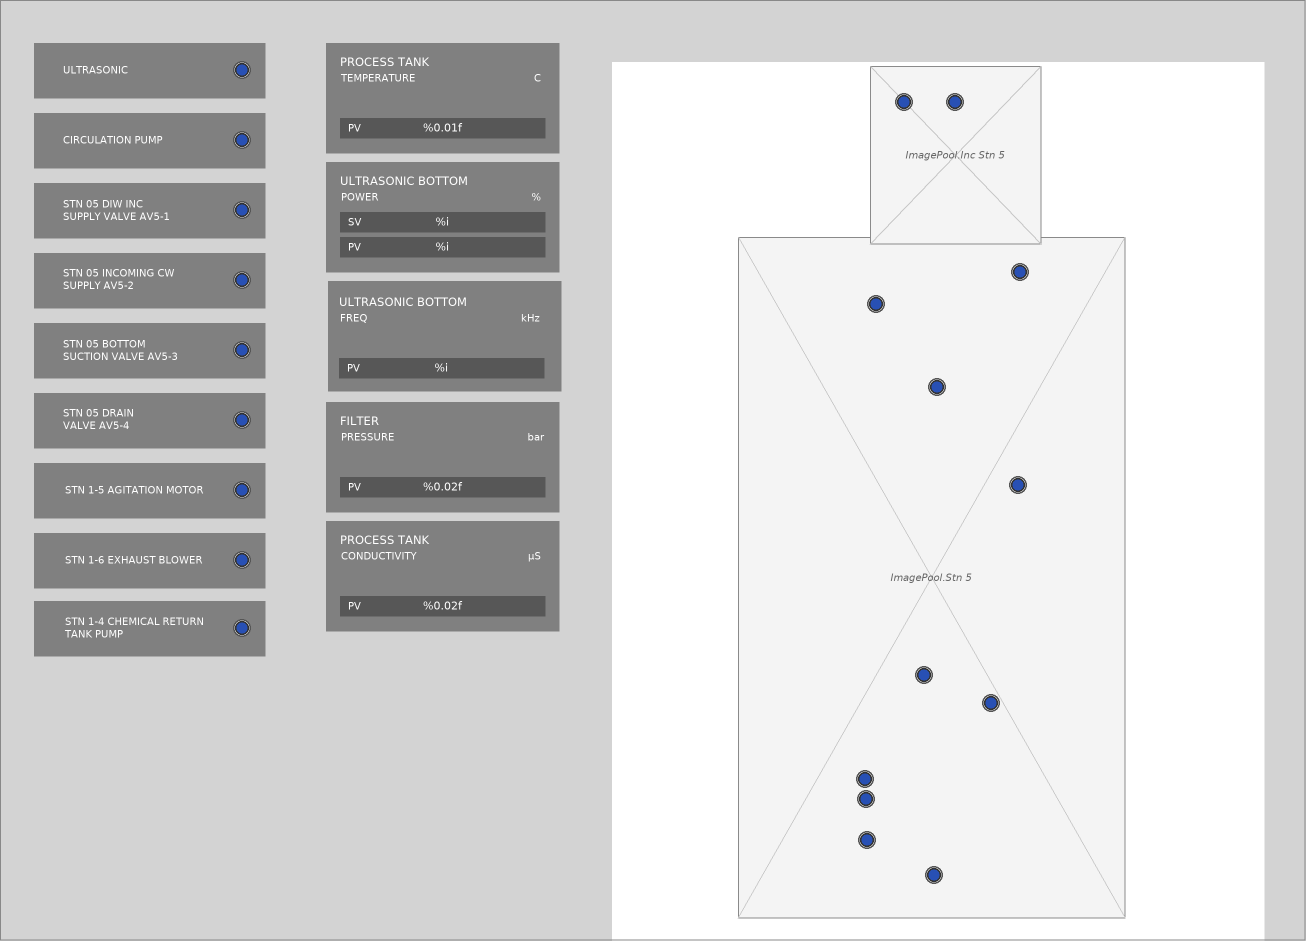
VISUALIZATION Auto_Station05  // 1306x941
    Rectangle (0,0 1306x875)
    RoundedRectangle (34,43 231x55)
    Label (60,62 163x16), "ULTRASONIC"
    Lamp1 (232,60 20x20), variable: ARdsMAP_HmiVariableStn[5].bProTankUsBtm_IND, style: Lamp-Lamp1-Blue
    RoundedRectangle (34,113 231x55)
    Label (60,132 151x16), "CIRCULATION PUMP"
    Lamp1 (232,130 20x20), variable: ARdsMAP_HmiVariableStn[5].bProTankPump_IND, style: Lamp-Lamp1-Blue
    RoundedRectangle (326,43 233x110)
    Label (337,54 150x16), "PROCESS TANK"
    Label (338,67 99x22), "TEMPERATURE"
    Label (515,67 29x22), "C"
    Label (345,92 22x22)
    Rectangle (340,118 205x20), "%0.01f", text variable: ARrStnTempPV[5]
    Label (345,117 22x22), "PV"
    Group (326,162 233x110)
        RoundedRectangle (0,0 233x110)
        Label (11,11 150x16), "ULTRASONIC BOTTOM"
        Label (12,24 99x22), "POWER"
        Label (189,24 29x22), "%"
        Rectangle (14,50 205x20), "%i", text variable: DSWeberEnclosure[1].DSWeberGenerator[3].IN_iTargetPowerPercentSetPoint
        Label (19,49 22x22), "SV"
        Rectangle (14,75 205x20), "%i", text variable: ARiStnUSBtmAPv[5]
        Label (19,74 22x22), "PV"
    RoundedRectangle (326,402 233x110)
    Label (337,413 150x16), "FILTER"
    Label (338,426 99x22), "PRESSURE"
    Label (515,426 32x22), "bar"
    Rectangle (340,477 205x20), "%0.02f", text variable: ARrStnFilterPressurePV[5]
    Label (345,476 22x22), "PV"
    RoundedRectangle (326,521 233x110)
    Label (337,532 150x16), "PROCESS TANK"
    Label (338,545 99x22), "CONDUCTIVITY"
    Label (515,545 29x22), "μS"
    Label (345,570 22x22)
    Rectangle (340,596 205x20), "%0.02f", text variable: ARrStnConductivityPV[5]
    Label (345,595 22x22), "PV"
    RoundedRectangle (328,281 233x110)
    Label (337,307 99x22), "FREQ"
    Label (336,294 150x16), "ULTRASONIC BOTTOM"
    Label (514,307 29x22), "kHz"
    Rectangle (339,358 205x20), "%i", text variable: ARiStnUSBtmAFreqPv[5]
    Label (344,357 22x22), "PV"
    RoundedRectangle (34,183 231x55)
    Label (60,197 151x27), "STN 05 DIW INC SUPPLY VALVE AV5-1"
    Lamp1 (232,200 20x20), variable: ARdsMAP_HmiVariableStn[5].bValve01_IND, style: Lamp-Lamp1-Blue
    RoundedRectangle (34,253 231x55)
    Lamp1 (232,270 20x20), variable: ARdsMAP_HmiVariableStn[5].bValve02_IND, style: Lamp-Lamp1-Blue
    Label (60,266 168x27), "STN 05 INCOMING CW SUPPLY AV5-2"
    RoundedRectangle (34,323 231x55)
    Label (60,337 151x27), "STN 05 BOTTOM SUCTION VALVE AV5-3"
    Lamp1 (232,340 20x20), variable: ARdsMAP_HmiVariableStn[5].bValve03_IND, style: Lamp-Lamp1-Blue
    RoundedRectangle (34,393 231x55)
    Lamp1 (232,410 20x20), variable: ARdsMAP_HmiVariableStn[5].bValve04_IND, style: Lamp-Lamp1-Blue
    Label (60,406 168x27), "STN 05 DRAIN VALVE AV5-4"
    RoundedRectangle (34,463 231x55)
    Label (62,472 160x36), "STN 1-5 AGITATION MOTOR"
    Lamp1 (232,480 20x20), variable: ARdsMAP_HmiVariableGeneral.bProTankAgitationMotor_IND, style: Lamp-Lamp1-Blue
    RoundedRectangle (34,533 231x55)
    Label (62,542 160x36), "STN 1-6 EXHAUST BLOWER"
    Lamp1 (232,550 20x20), variable: ARdsMAP_HmiVariableGeneral.bExhaustBlower_IND, style: Lamp-Lamp1-Blue
    RoundedRectangle (34,601 231x55)
    Label (62,610 160x36), "STN 1-4 CHEMICAL RETURN TANK PUMP"
    Lamp1 (232,618 20x20), variable: ARdsMAP_HmiVariableGeneral.bProTankPump_IND, style: Lamp-Lamp1-Blue
    Rectangle (612,62 652x879)
    Image (738,237 387x681), image: ImagePool.Stn 5
    Lamp1 (927,377 20x20), variable: ARdsMAP_HmiVariableStn[5].bProTankUsBtm_IND, style: Lamp-Lamp1-Blue
    Lamp1 (914,665 20x20), variable: ARdsMAP_HmiVariableStn[5].bProTankPump_IND, style: Lamp-Lamp1-Blue
    Lamp1 (981,693 20x20), variable: ARdsMAP_HmiVariableStn[5].bValve04_IND, style: Lamp-Lamp1-Blue
    Lamp1 (1008,475 20x20), variable: ARdsMAP_HmiVariableStn[5].bValve03_IND, style: Lamp-Lamp1-Blue
    Lamp1 (866,294 20x20), variable: ARdsMAP_HmiVariableStn[5].bProcessTankMinLevel_IND, style: Lamp-Lamp1-Blue
    Lamp1 (1010,262 20x20), variable: ARdsMAP_HmiVariableStn[5].bOverflowMaxLevel_IND, style: Lamp-Lamp1-Blue
    Lamp1 (857,830 20x20), variable: ARdsMAP_HmiVariableStn[5].bSubTankMinLevel_IND, style: Lamp-Lamp1-Blue
    Lamp1 (856,789 20x20), variable: ARdsMAP_HmiVariableStn[5].bSubTankRegLevel_IND, style: Lamp-Lamp1-Blue
    Lamp1 (855,769 20x20), variable: ARdsMAP_HmiVariableStn[5].bSubTankMaxLevel_IND, style: Lamp-Lamp1-Blue
    Lamp1 (924,865 20x20), variable: ARdsMAP_HmiVariableGeneral.bProTankPump_IND, style: Lamp-Lamp1-Blue
    Image (870,66 171x178), image: ImagePool.Inc Stn 5
    Lamp1 (894,92 20x20), variable: ARdsMAP_HmiVariableStn[5].bValve01_IND, style: Lamp-Lamp1-Blue
    Lamp1 (945,92 20x20), variable: ARdsMAP_HmiVariableStn[5].bValve02_IND, style: Lamp-Lamp1-Blue
END_VISUALIZATION

(* stored: Version 1.1.0.1, ProductVersion 3.1.4024.12
   Visu Auto_Station05: Id {0cd9057b-f866-48eb-8a3e-b0ec08d67b05} *)
